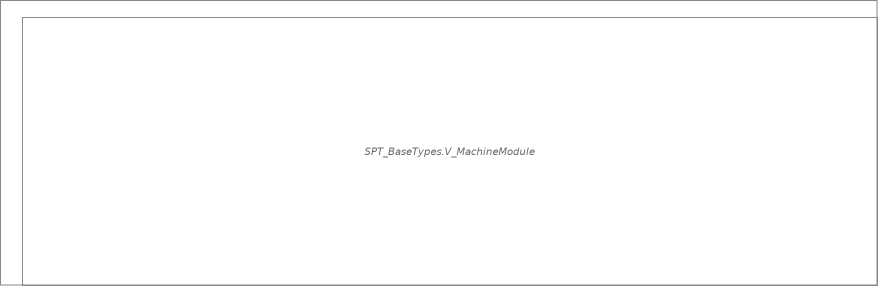
VISUALIZATION Visualization  // 878x286
    Frame (22,17 856x269)
        shows SPT_BaseTypes.V_MachineModule(HMI := MAIN.Machine.PackMLBaseModule_HMI)
END_VISUALIZATION

(* stored: Version 1.1.0.1, ProductVersion 3.1.4024.12
   Visu Visualization: Id {3c1070b5-750b-48ca-a34d-b27b9f1c5010} *)
